Fanuc KAREL source: kc00001.KL

-- PROVISIONAL review KL for V940-1; original PC SHA256 0b5f09fc7fa3ac2999db6cb32d1ba91c03618785aabdff07f8bd504c112d4419
-- Incomplete behavior may be omitted. Consult companion uncertainty JSON. Do not deploy.
PROGRAM KC00001
%NOLOCKGROUP
BEGIN
  -- V9_ZERO_TABLE_METADATA_HINT layout=0002_ascii; no indexed target words; source/name/runtime held
  -- UNRESOLVED_PC offsets 5-14; opcodes 3F,75
  -- UNRESOLVED_PC offsets 19-28; opcodes 3F,75
  -- UNRESOLVED_PC offsets 33-71; opcodes 27,22,22,22,2A,22,2A,22,31
  -- UNRESOLVED_PC offsets 76-80; opcodes 7F
END KC00001
